PROGRAM MAIN
VAR
	counter : INT := 0;
END_VAR

counter := counter + 1;
GVL.global_counter := GVL.global_counter + 1;

END_PROGRAM

(* stored: Version 1.1.0.1, ProductVersion 3.1.4024.15
   POU MAIN: Id {37e4aa0d-7777-400c-a8ca-388435fd5c5b}, SpecialFunc None *)
